// TIA Portal project "BloqueFuncionFB" (V16)

(* hardware
DEVICE "S7-1200 station_1"  S7-1200 Station
   slot 0: "Rack_0"  S7-1200 Rack  Rack  V1.0
   slot 1: "PLC_1"  CPU 1214C AC/DC/Rly  6ES7 214-1BG40-0XB0  V4.4
*)

// ===== PLC "PLC_1"  CPU 1214C AC/DC/Rly =====

VAR_GLOBAL   // PLC tag table "Tabla de variables estándar"
   ""Tag_1"" AT %I1.0 : Bool;
   ""Tag_2"" AT %I1.1 : Bool;
   ""Tag_4"" AT %I1.2 : Bool;
   ""Tag_5"" AT %I1.3 : Bool;
   ""Tag_7"" AT %I1.4 : Bool;
   ""Tag_8"" AT %I1.5 : Bool;
   ""Tag_3"" AT %Q1.0 : Bool;
   ""Tag_6"" AT %Q1.1 : Bool;
   ""Tag_9"" AT %Q1.2 : Bool;
END_VAR